Yaskawa INFORM job: DXF_Prueba20250507162858.JBI

/JOB
//NAME DXF_Prueba20250507162858
//POS
///NPOS 5,0,0,0,0,0
///TOOL 0
///POSTYPE PULSE
///PULSE
C00000=0,0,0,0,0,0
C00001=50000,0,5000,0,0,0
C00002=50000,-50000,5000,0,0,0
C00003=0,-50000,5000,0,0,0
C00004=0,0,5000,0,0,0
//INST
///DATE 2025/05/07 16:28
///ATTR SC,RW
///GROUP1 RB1
NOP
MOVJ C00000 VJ=10.0
MOVL C00001 V=10.0
MOVL C00002 V=10.0
MOVL C00003 V=10.0
MOVL C00004 V=10.0
END
